FUNCTION_BLOCK Ps10Axis EXTENDS AxesBase
VAR_INPUT
END_VAR
VAR_OUTPUT
END_VAR
VAR
	{attribute 'OPC.UA.DA' := '0'}
	_config : Ps10OwisAxisConfig;
	{attribute 'OPC.UA.DA' := '0'}
	_coeAccess : CoeAccess;
	{attribute 'OPC.UA.DA' := '0'}
	_initConfigSerialCom : BOOL;	
	{attribute 'OPC.UA.DA' := '0'}
	_serialCom  : SerialCom(Prefix :='', Suffix := Const.CARRIAGE_RETURN);
	{attribute 'OPC.UA.DA' := '0'}
	_refSerialCom : REFERENCE TO SerialCom(Prefix :='', Suffix := Const.CARRIAGE_RETURN) := _serialCom;	 
	{attribute 'OPC.UA.DA' := '0'}
	_isReceived : BOOL;
	
	{attribute 'OPC.UA.DA' := '0'}
	_deliverMessages : INT;
	
	StatusMsg : STRING(255);
	AxisStatusMsg : STRING(255);
	DrivingCurrentMsg : STRING(255);
	HoldingCurrentMsg : STRING(255);
	LimitSwitchtMsg : STRING(255);
	ErrMsg : STRING(255);
	PositionMsg : STRING(255);
	CustomMsg : STRING(255);
	IsInMovingMsg : STRING(255);
	
	{region 'Commands'}	

	{attribute 'OPC.UA.DA' := '0'}
	_cmdConfigDeviceParameters : BOOL;
	{attribute 'OPC.UA.DA' := '0'}
	_cmdClearErr : BOOL;
	{attribute 'OPC.UA.DA' := '0'}
	_cmdMotorInit : BOOL;
	{attribute 'OPC.UA.DA' := '0'}
	_cmdDrivingCurrent : BOOL;
	{attribute 'OPC.UA.DA' := '0'}
	_cmdHoldingCurrent : BOOL;
	{attribute 'OPC.UA.DA' := '0'}	 
	_cmdLimitSwitch : BOOL;
	{attribute 'OPC.UA.DA' := '0'}
	_cmdReset : BOOL;
	{attribute 'OPC.UA.DA' := '0'}
	_cmdStopMotion : BOOL;		 
	{attribute 'OPC.UA.DA' := '0'}
	_cmdHomePosition : BOOL;
	{attribute 'OPC.UA.DA' := '0'}
	_cmdMoveAbsPosition : BOOL;
	{attribute 'OPC.UA.DA' := '0'}
	_customCmd : BOOL;
	{attribute 'OPC.UA.DA' := '0'}			  		   
	_cmdRaiseProperties : BOOL;	 
			
	{endregion}
		 
	{attribute 'OPC.UA.DA' := '0'}
	_initDevice : BOOL;	
		
	{attribute 'OPC.UA.DA' := '0'}
	_posToDegree : LREAL;
	{attribute 'OPC.UA.DA' := '0'}
	_cmd : STRING;
	{attribute 'OPC.UA.DA' := '0'}
	_itemScheduler : INT;
	{attribute 'OPC.UA.DA' := '0'}
	_itemRaisedProperties : INT;
	{attribute 'OPC.UA.DA' := '0'}
	_itemMove : INT;	
	{attribute 'OPC.UA.DA' := '0'}
	_itemInit : INT;
	{attribute 'OPC.UA.DA' := '0'}
	_itemdConfigDeviceParameters : INT;
	{attribute 'OPC.UA.DA' := '0'}
	_pulseGenerator : TON;
	{attribute 'OPC.UA.DA' := '0'}
	_pulseMoveGenerator : TON;	
	{attribute 'OPC.UA.DA' := '0'}
	_initPulseGenerator : TON;	
	{attribute 'OPC.UA.DA' := '0'}	
	_execPulseGenerator : TON;
	{attribute 'OPC.UA.DA' := '0'}	
	_configDeviceParamsPulseGenerator : TON;	
	
	{attribute 'OPC.UA.DA' := '0'}
	message : STRING;
	{attribute 'OPC.UA.DA' := '0'}
	lastMessage : STRING;	
	{attribute 'OPC.UA.DA' := '0'}
	stringLength : INT;
	{attribute 'OPC.UA.DA' := '0'}
	_convertDegreeToCount : LREAL := 83;
	{attribute 'OPC.UA.DA' := '0'}
	_currentAxisMode : STRING;
	{attribute 'OPC.UA.DA' := '0'}
	_currentPos : LREAL;	
	{attribute 'OPC.UA.DA' := '0'} 
	_currentPositionCounter : UINT;
	{attribute 'OPC.UA.DA' := '0'} 
	_isInMoving : BOOL;
END_VAR

IF NOT InitConfigSerialCom THEN
	ConfigureSerialCom();
ELSIF THIS^.Status = TExecutionState.Ready THEN				
	IF _refSerialCom.ErrorReceiveId = COMERROR_NOERROR THEN
		_refSerialCom(TxBuffer:= HardwareGlobalVariables.TxBufferFilterWheel, 
		 	      	  RxBuffer:= HardwareGlobalVariables.RxBufferFilterWheel);
	END_IF			

	// Init device	
	InitDevice();
		 				  	
	// Deliver messages
	IF _refSerialCom.IsReceived THEN		
		lastMessage := _refSerialCom.LastReceivedString;			
		stringLength := LEN(lastMessage);
		
		IF stringLength > 1 THEN
			message := LEFT(lastMessage, stringLength - 1);
		ELSE
			message := ' ';
		END_IF; 
				
		CASE _deliverMessages OF	
			EFeedbackMsgOwisPs10.AxisStateMsg :
				_currentAxisMode := MID(message, 1, STRING_TO_INT(AxesConst.AXIS_FILTER_WHEEL));
				AxisStatusMsg := ParseAxisStatus(_currentAxisMode);
			EFeedbackMsgOwisPs10.DrivingCurrentMsg :
				 DrivingCurrentMsg := message;
			EFeedbackMsgOwisPs10.HoldingCurrentMsg :
				 HoldingCurrentMsg := message;
			EFeedbackMsgOwisPs10.LimitSwitchMsg :
				 LimitSwitchtMsg := message;
			EFeedbackMsgOwisPs10.ErrMsg :
				 ErrMsg := message;
			EFeedbackMsgOwisPs10.PositionMsg :					
				_currentPos := STRING_TO_LREAL(message) / _convertDegreeToCount;
				PositionMsg := LREAL_TO_STRING(_currentPos);				
			EFeedbackMsgOwisPs10.CurrentPositionCounterMsg :
				_currentPositionCounter := STRING_TO_UINT(message);			
			EFeedbackMsgOwisPs10.CustomMsg :
				CustomMsg := message;						
			END_CASE
	END_IF		
			
	IF (_initDevice AND NOT _cmdClearErr AND NOT _cmdMotorInit AND NOT _cmdConfigDeviceParameters AND NOT _cmdDrivingCurrent AND NOT 
		_cmdHoldingCurrent AND NOT _cmdLimitSwitch AND NOT _cmdStopMotion AND NOT _cmdHomePosition AND NOT _cmdMoveAbsPosition AND NOT 
		_customCmd AND NOT _cmdRaiseProperties) THEN
			MessageScheduler();
	END_IF
	
	ConfigDeviceParameters(_cmdConfigDeviceParameters);
	ClearError(_cmdClearErr);
	MotorInit(_cmdMotorInit);
	SetDrivingCurrent(_cmdDrivingCurrent);
	SetHoldingCurrent(_cmdHoldingCurrent);
	SetLimitSwitch(_cmdLimitSwitch);
	Reset(_cmdReset);
	StopMotion(_cmdStopMotion);
	HomePosition(_cmdHomePosition);	
	MoveAbsPosition(_cmdMoveAbsPosition, _posToDegree);
	CustomCommand(_customCmd, _cmd);	
	RaisePropertiesChanged(_cmdRaiseProperties);	
	
END_IF

{attribute 'TcRpcEnable' := '1'}
METHOD ClearError
VAR_INPUT
	Execute : BOOL;
END_VAR
VAR
	cmd : STRING := 'ERRCLEAR';
END_VAR
IF Execute THEN
	_logger.Information(_message.Reset().Append(_config.Name).Append(' - Clear error').ToString());
	_serialCom.Send(cmd);	

	_cmdClearErr := FALSE;
END_IF
END_METHOD

METHOD ConfigDeviceParameters
VAR_INPUT
	Execute : BOOL;
END_VAR
VAR	
END_VAR
IF Execute THEN

	_cmdConfigDeviceParameters := TRUE;	

	IF _configDeviceParamsPulseGenerator.Q THEN
		_configDeviceParamsPulseGenerator(IN := FALSE, PT := T#10MS);
		
		CASE _itemdConfigDeviceParameters OF
			0:  _logger.Information(_message.Reset().Append(_config.Name).Append(' - Configure device parameters').ToString());
				_itemdConfigDeviceParameters := 1;				
								
			1: _cmdDrivingCurrent := TRUE;
				_itemdConfigDeviceParameters := 2;

			2: _cmdHoldingCurrent := TRUE;
				_itemdConfigDeviceParameters := 3;				
			
			3: _cmdLimitSwitch := TRUE;
				_itemdConfigDeviceParameters := 4;	
			
			4: _cmdMotorInit := TRUE;
				_itemdConfigDeviceParameters := 5;					
				
			5: _logger.Information(_message.Reset(). Append(_config.Name). Append(' - Configure device parameters done').ToString());	
			   _itemdConfigDeviceParameters := 0;			
			   _cmdConfigDeviceParameters := FALSE;
		END_CASE
	ELSE
		_configDeviceParamsPulseGenerator(IN := TRUE, PT := T#200MS);		
	END_IF		
END_IF
END_METHOD

METHOD ConfigureSerialCom
VAR_INPUT
END_VAR
IF _coeAccess.CoeOperation.Ready THEN
	_logger.Information(_message.Reset().Append('Start configuration com serial').ToString());
END_IF;	

_coeAccess.CoeOperation.Start();
_coeAccess(SerialCommunication := _config.SerialCommunication);
	
IF _coeAccess.CoeOperation.Done THEN
	_coeAccess.SetDone();	
 
	_Logger.Information(_message.Reset().
							Append('{').Append(TO_STRING(THIS^.Family)).Append('} : ').
							Append(' - Status : ').Append(TO_STRING(_coeAccess.Status)).ToString());	
	InitConfigSerialCom := TRUE;
END_IF
 
IF _coeAccess.CoeOperation.Error THEN	
	_coeAccess.SetError(0);
	
	_Logger.Error(_message.Reset().
							Append('{').Append(TO_STRING(THIS^.Family)).Append('} : ').
							Append(' - Status : ').Append(TO_STRING(_coeAccess.Status)).ToString());
	InitConfigSerialCom := TRUE;
END_IF

THIS^.Status := _coeAccess.Status;
State := _coeAccess.Status;
END_METHOD

{attribute 'TcRpcEnable' := '1'}
METHOD CustomCommand
VAR_INPUT
	Execute : BOOL;
	Cmd : STRING;
END_VAR
IF Execute THEN
	_logger.Information(_message.Reset().Append(_config.Name).Append(' - Custom : ').Append(Cmd).ToString());
	_deliverMessages := EFeedbackMsgOwisPs10.CustomMsg;									
	_serialCom.Send(Cmd);
	
	_customCmd := FALSE;
END_IF
END_METHOD

{attribute 'TcRpcEnable' := '1'}
METHOD ErrorMessages
VAR_INPUT
END_VAR
VAR
	cmd : STRING := '?MSG';
END_VAR
_deliverMessages := EFeedbackMsgOwisPs10.ErrMsg;	
_serialCom.Send(cmd);
END_METHOD

METHOD FB_init : BOOL
VAR_INPUT
	bInitRetains : BOOL; // if TRUE, the retain variables are initialized (warm start / cold start)
	bInCopyCode : BOOL;  // if TRUE, the instance afterwards gets moved into the copy code (online change)
	Config : Ps10OwisAxisConfig;
END_VAR
IF Config.IsEnabled THEN
	_config := Config;
	
	SUPER^._axisConfig.Name := Config.Name;
	SUPER^._axisConfig.DeviceID := Config.DeviceID;
	SUPER^._axisConfig.IsEnabled := Config.IsEnabled;
	SUPER^._axisConfig.LogLevel := Config.LogLevel;
	
	SUPER^.Name := Config.Name;
	SUPER^.DeviceID := Config.DeviceID;	
	THIS^.Family := DeviceFamily.Axes;
	
	_Logger.Information(_message.Reset().Append('Init ').
							Append('{').Append(TO_STRING(THIS^.Family)).Append('} - ').
							Append('{').Append(TO_STRING(Config.Name)).Append('}').ToString());																													
END_IF
END_METHOD

(** Axis state inquiry **)
METHOD GetAxisStatus : STRING
VAR_INPUT
END_VAR
VAR
	cmd : STRING := '?ASTAT';
END_VAR
_deliverMessages := EFeedbackMsgOwisPs10.AxisStateMsg;	
_serialCom.Send(cmd);
END_METHOD

(** Read out driving current with stepper motors in percent **)
METHOD PROTECTED GetDrivingCurrent
VAR_INPUT
END_VAR
VAR
	cmd : STRING := '?DRICUR';
END_VAR
_deliverMessages := EFeedbackMsgOwisPs10.DrivingCurrentMsg;	
_serialCom.Send(Concat(cmd, AxesConst.AXIS_FILTER_WHEEL));
END_METHOD

(** Read out holding current with stepper motor axis in percent **)
METHOD PROTECTED GetHoldingCurrent
VAR_INPUT
END_VAR
VAR
	cmd : STRING := '?HOLCUR';
END_VAR
_deliverMessages := EFeedbackMsgOwisPs10.HoldingCurrentMsg;	
_serialCom.Send(Concat(cmd, AxesConst.AXIS_FILTER_WHEEL));
END_METHOD

(** Read out limit switch mask for the axis **)
METHOD PROTECTED GetLimitSwitch
VAR_INPUT
END_VAR
VAR
	cmd : STRING := '?SMK';
END_VAR
_deliverMessages := EFeedbackMsgOwisPs10.LimitSwitchMsg;	
_serialCom.Send(Concat(cmd, AxesConst.AXIS_FILTER_WHEEL));
END_METHOD

(** Position Query **)
METHOD PROTECTED GetPosition
VAR_INPUT
END_VAR
VAR
	cmd : STRING := '?PSET';
END_VAR
_deliverMessages := EFeedbackMsgOwisPs10.PositionMsg;	
_serialCom.Send(Concat(cmd, AxesConst.AXIS_FILTER_WHEEL));
END_METHOD

{attribute 'TcRpcEnable' := '1'}
METHOD HomePosition
VAR_INPUT
	Execute : BOOL;
END_VAR
VAR
	cmd : STRING := 'REF';
END_VAR
IF Execute THEN	
	_logger.Information(_message.Reset().Append(_config.Name).Append(' - Home position : ').ToString());
	cmd := Concat(CONCAT(cmd, AxesConst.AXIS_FILTER_WHEEL), '=');	
	_serialCom.Send(Concat(cmd, '4'));
	
	_cmdHomePosition := FALSE;
END_IF
END_METHOD

PROPERTY InitConfigSerialCom : BOOL
GET
InitConfigSerialCom := _initConfigSerialCom;
END_GET
SET
_initConfigSerialCom := InitConfigSerialCom;
END_SET
END_PROPERTY

METHOD InitDevice
VAR_INPUT
END_VAR
VAR
	displayingPositionCmd : STRING := 'PWMSMODE';
	absoluteModeCmd : STRING := 'ABSOL';
	
	displayingPositionInDegree : STRING;
END_VAR
IF NOT _initDevice THEN	
	IF _initPulseGenerator.Q THEN
		_initPulseGenerator(IN := FALSE, PT := T#10MS);
		
		CASE _itemInit OF
			0:  _logger.Information(_message.Reset().Append(_config.Name).Append(' - InitDevice').ToString());
				_itemInit := 1;				
				
			1:  _cmdClearErr := TRUE;
				_itemInit := 2;
			
			2: // Absolute mode
				_serialCom.Send(CONCAT(absoluteModeCmd, AxesConst.AXIS_FILTER_WHEEL));	
				_itemInit := 10;
				
			10: _cmdConfigDeviceParameters := TRUE;	
			   _itemInit := 11;
			
			11: IF NOT _cmdConfigDeviceParameters THEN
					_itemInit := 20;
				END_IF
			
			20: GetAxisStatus();
				_itemInit := 21;
				
			21: // Displaying position in °
				displayingPositionInDegree := Concat(CONCAT(displayingPositionCmd, AxesConst.AXIS_FILTER_WHEEL), '=');
				_serialCom.Send(CONCAT(displayingPositionInDegree, '3'));				
				_itemInit := 22;													
				
			22:  IF _currentAxisMode = 'R' THEN	
					_itemInit := 30;	
				ELSE			
					_logger.Error(_message.Reset().Append(_config.Name).Append(' - Axis status : ').
								  Append(_currentAxisMode).ToString());
					_itemInit := 40;				  
			    END_IF							
				
			30:  GetPosition();
				_itemInit := 31;	
				
			31: _posToDegree := _currentPos;
				_itemInit := 40;
				
			40: _logger.Information(_message.Reset(). Append(_config.Name). Append(' - InitDevice done').ToString());	
				_itemInit := 0;			
				_initDevice	:= TRUE;
		END_CASE
	ELSE
		_initPulseGenerator(IN := TRUE, PT := T#100MS);		
	END_IF		
END_IF
END_METHOD

PROPERTY IsInMoving : bool
GET
IsInMoving := _isInMoving;
END_GET
SET
_isInMoving := IsInMoving;
END_SET
END_PROPERTY

METHOD MessageScheduler
VAR_INPUT
END_VAR
IF _pulseGenerator.Q THEN
	_pulseGenerator(IN := FALSE, PT := T#10MS);
	
	CASE _itemScheduler OF				
		0:	GetAxisStatus();
			_itemScheduler := 1;
						
		1:	GetPosition();
			_itemScheduler := 0;			
	END_CASE		
ELSE
	_pulseGenerator(IN := TRUE, PT := T#100MS);		
END_IF
END_METHOD

{attribute 'TcRpcEnable' := '1'}
METHOD MotorInit
VAR_INPUT
	Execute : BOOL;
END_VAR
VAR	
	cmd : STRING := 'INIT';
END_VAR
IF Execute THEN
	_logger.Information(_message.Reset().Append(_config.Name).Append(' - Enable the motor power stage').ToString());
	_serialCom.Send(Concat(cmd, AxesConst.AXIS_FILTER_WHEEL));	

	_cmdMotorInit := FALSE;	
END_IF
END_METHOD

{attribute 'TcRpcEnable' := '1'}
METHOD PROTECTED MoveAbsPosition 
VAR_INPUT
	Execute : BOOL;
	Position : LREAL;
END_VAR
VAR
	cmdSet : STRING := 'PSET';
	cmdGo : STRING := 'PGO';
	cmdCnt : STRING := '?CNT';
	cmd : STRING;	
END_VAR
IF Execute THEN

	_cmdMoveAbsPosition := TRUE;
	_posToDegree := Position;	
	
	IF _pulseMoveGenerator.Q THEN
		_pulseMoveGenerator(IN := FALSE, PT := T#10MS);
	
		CASE _itemMove OF
			0:	_logger.Information(_message.Reset().Append(_config.Name).Append(' - Move absolute position : ').
													 Append(TO_STRING(_posToDegree)).Append(' °').ToString());
								
				cmd := Concat(CONCAT(cmdSet, AxesConst.AXIS_FILTER_WHEEL), '=');				
				_serialCom.Send(CONCAT(cmd, LREAL_TO_STRING(_posToDegree * _convertDegreeToCount)));				
				_itemMove := 1;						
				
			1:  _serialCom.Send(Concat(cmdGo, AxesConst.AXIS_FILTER_WHEEL));											
				_itemMove := 2;	
				
			2:  _deliverMessages := EFeedbackMsgOwisPs10.CurrentPositionCounterMsg;	
				IF _currentPositionCounter <> (_posToDegree * _convertDegreeToCount) THEN					
					_serialCom.Send(Concat(cmdCnt, AxesConst.AXIS_FILTER_WHEEL));
					IsInMovingMsg := BOOL_TO_STRING(TRUE);	
				ELSE
					IsInMovingMsg := BOOL_TO_STRING(FALSE);	
					_itemMove := 3;	
				END_IF
								
			3: _cmdMoveAbsPosition := FALSE;
				_itemMove := 0;
			
		END_CASE			
	ELSE
		_pulseMoveGenerator(IN := TRUE, PT := T#100MS);	
	END_IF

END_IF
END_METHOD

METHOD PRIVATE ParseAxisStatus : STRING
VAR_INPUT
	CurrentAxisMode : STRING;
END_VAR
VAR
	Description : STRING;
END_VAR
IF CurrentAxisMode = 'I' THEN
	Description := 'Axis is not initialized';
ELSIF CurrentAxisMode = 'O' THEN
	Description := 'Axis is disabled';
ELSIF CurrentAxisMode = 'R' THEN
	Description := 'Axis initialized and ready';
ELSIF CurrentAxisMode = 'T' THEN
	Description := 'Axis is positioning in trapezoidal profile';
ELSIF CurrentAxisMode = 'V' THEN
	Description := 'Axis is operating in velocity mode';
ELSIF CurrentAxisMode = 'P' THEN
	Description := 'Reference motion is in progress';
ELSIF CurrentAxisMode = 'F' THEN
	Description := 'Axis is releasing a limit switch';
ELSIF CurrentAxisMode = 'L' THEN
	Description := 'Axis has been disabled after approaching a hardware limit switch(MINSTOP, MAXSTOP)';
ELSIF CurrentAxisMode = 'B' THEN
	Description := 'Aaxis has been stopped after approaching a brake switch(MINDEC, MAXDEC)';
ELSIF CurrentAxisMode = 'A' THEN
	Description := 'Axis has been disabled after limit switch error';
ELSIF CurrentAxisMode = 'M' THEN
	Description := 'Axis has been disabled after motion-controller error';
ELSIF CurrentAxisMode = 'Z' THEN
	Description := 'Axis has been disabled after timeout error';
ELSIF CurrentAxisMode = 'H' THEN
	Description := 'Phase initialization active (step motor axis)';
ELSIF CurrentAxisMode = 'U' THEN
	Description := 'Axis not enabled';
ELSIF CurrentAxisMode = 'E' THEN
	Description := 'Axis has been disabled after motion error';
ELSIF CurrentAxisMode = '?' THEN
	Description := 'Error, unknown state of axis';
ELSE
	Description := 'Unknown error';
END_IF

ParseAxisStatus := Description;
END_METHOD

{attribute 'TcRpcEnable' := '1'}
METHOD RaisePropertiesChanged
VAR_INPUT
	Execute : BOOL;
END_VAR
IF Execute THEN
	IF THIS^.Status <> TExecutionState.Ready THEN	
		_cmdRaiseProperties := FALSE;
		RETURN;
	END_IF	

	_cmdRaiseProperties := TRUE;
	
	IF _pulseGenerator.Q THEN
		_pulseGenerator(IN := FALSE, PT := T#10MS);	

		CASE _itemRaisedProperties OF
			0:  StateMsg := ' ';
				AxisStatusMsg := ' ';
				ErrMsg := ' ';
				PositionMsg := ' ';
				CustomMsg := ' ';
				
				_itemRaisedProperties := 10;
			
			10:  GetPosition();
				_itemRaisedProperties := 11;
			
			11:  GetAxisStatus();
				 _itemRaisedProperties := 12;
				 
			12:  ErrorMessages();
				 _itemRaisedProperties := 20;			
				 
			20:  _logger.Information(_message.Reset().Append(_config.Name).Append(' - PS10 Axis RaisePropertiesChanged').ToString());
				_cmdRaiseProperties := FALSE;				
				_itemRaisedProperties := 0;
			
		END_CASE
	ELSE
		_pulseGenerator(IN := TRUE, PT := T#100MS);	
	END_IF
END_IF
END_METHOD

{attribute 'TcRpcEnable' := '1'}
METHOD Reset
VAR_INPUT
	Execute : BOOL;
END_VAR
VAR
	cmd : STRING := 'RESETMB';
END_VAR
IF Execute THEN
	_logger.Information(_message.Reset().Append(_config.Name).Append(' - Release reset main board').ToString());
	_serialCom.Send(cmd);	
	
	_cmdReset := FALSE;
END_IF
END_METHOD

{attribute 'TcRpcEnable' := '1'}
METHOD SetDrivingCurrent
VAR_INPUT
	Execute : BOOL;
END_VAR
VAR
	cmdSet : STRING := 'DRICUR';
	cmd : STRING;
END_VAR
IF Execute THEN
	_logger.Information(_message.Reset().Append(_config.Name).Append(' - driving current with stepper motor: ').
		Append(TO_STRING(AxesConst.FW_DRIVING_CURRENT_IN_PERCENT)).ToString());
	
	cmd := Concat(CONCAT(cmdSet, AxesConst.AXIS_FILTER_WHEEL), '=');
	_serialCom.Send(CONCAT(cmd, TO_STRING(AxesConst.FW_DRIVING_CURRENT_IN_PERCENT)));	

	_cmdDrivingCurrent := FALSE;	
END_IF
END_METHOD

{attribute 'TcRpcEnable' := '1'}
METHOD SetHoldingCurrent
VAR_INPUT
	Execute : BOOL;
END_VAR
VAR
	cmdSet : STRING := 'HOLCUR';
	cmd : STRING;
END_VAR
IF Execute THEN
	_logger.Information(_message.Reset().Append(_config.Name).Append(' - holding current with stepper motor axes: ').
		Append(TO_STRING(AxesConst.FW_HOLDING_CURRENT_IN_PERCENT)).ToString());
	
	cmd := Concat(CONCAT(cmdSet, AxesConst.AXIS_FILTER_WHEEL), '=');
	_serialCom.Send(CONCAT(cmd, TO_STRING(AxesConst.FW_HOLDING_CURRENT_IN_PERCENT)));	

	_cmdHoldingCurrent := FALSE;	
END_IF
END_METHOD

{attribute 'TcRpcEnable' := '1'}
METHOD SetLimitSwitch
VAR_INPUT
	Execute : BOOL;
END_VAR
VAR
	cmdSet : STRING := 'SMK';
	cmd : STRING;
END_VAR
IF Execute THEN
	_logger.Information(_message.Reset().Append(_config.Name).Append(' -  limit switch mask for the axis: ').
		Append(TO_STRING(AxesConst.FW_LIMIT_SWITCH_MASK)).ToString());
	
	cmd := Concat(CONCAT(cmdSet, AxesConst.AXIS_FILTER_WHEEL), '=');
	_serialCom.Send(CONCAT(cmd, TO_STRING(AxesConst.FW_LIMIT_SWITCH_MASK)));	

	_cmdLimitSwitch := FALSE;	
END_IF
END_METHOD

{attribute 'TcRpcEnable' := '1'}
METHOD StopMotion
VAR_INPUT
	Execute : BOOL;
END_VAR
VAR
	cmd : STRING := 'STOP1';
END_VAR
IF Execute THEN	
	_logger.Information(_message.Reset().Append(_config.Name).Append(' - Stop motion').ToString());
	_serialCom.Send(cmd);
	
	_cmdStopMotion := FALSE;
END_IF
END_METHOD

END_FUNCTION_BLOCK

(* stored: Version 1.1.0.1, ProductVersion 3.1.4024.12
   POU Ps10Axis: Id {65318552-fa8a-4be4-9877-1eb5da08e2e6}, SpecialFunc None
   Folder Comamnds: Id {350d7b4c-9999-4614-8983-2b0788406443}
   Method ClearError: Id {9cf50f82-dedf-4020-a341-c2e03f9bd16b}
   Method ConfigDeviceParameters: Id {9dd7c1a3-38a3-4271-adf2-d5c1fd271f87}
   Method ConfigureSerialCom: Id {92ee4274-1822-4857-a351-1af2244cf04e}
   Method CustomCommand: Id {04426e00-f477-4383-857a-2ae2c5de4dbe}
   Method ErrorMessages: Id {af95c508-4de3-4b04-ad88-3fb38c9b4a6e}
   Method FB_init: Id {c9eecb17-8010-4deb-b770-2d445332fb7a}
   Method GetAxisStatus: Id {3fbf2da0-a10e-4662-ab0b-95ea943ad0ed}
   Method GetDrivingCurrent: Id {92b3f748-1524-4586-a2ca-ecd6e1233df8}
   Method GetHoldingCurrent: Id {1eac2e4b-31a7-47d1-83e9-91a91d90e56e}
   Method GetLimitSwitch: Id {d69a0b29-70d3-44d2-b788-e7ab365eced6}
   Method GetPosition: Id {55a3b673-e715-4d70-9fa7-5225e4770e89}
   Method HomePosition: Id {142d51a5-57ef-4f7b-b18a-4cfaf2920b91}
   Property InitConfigSerialCom: Id {2aa5b88d-df39-4f9b-949f-1e8e44a662c9}
   Get Get: Id {494cec2c-0a6e-4e21-8cea-50ca2358b100}
   Set Set: Id {5729c6bb-be11-4151-8251-605ad3510059}
   Method InitDevice: Id {5c2fcf27-05f4-4bb9-9c40-55e9bc5563c8}
   Property IsInMoving: Id {43f5a690-3f81-4021-9bd2-2250a324fef6}
   Get Get: Id {43b5b94b-ba0a-4053-90d8-b0b48186412a}
   Set Set: Id {5eefe730-1f7f-423f-84ac-5e9df6527cc9}
   Method MessageScheduler: Id {d15cb2a3-cb63-4708-a63c-d14e3c192308}
   Method MotorInit: Id {9d90297e-68a2-4beb-b5a0-edfb71b5534e}
   Method MoveAbsPosition: Id {e52af445-02be-4345-a161-7a76bf74adb8}
   Method ParseAxisStatus: Id {2ff9b0bb-a1ce-404f-9822-774a93978c34}
   Method RaisePropertiesChanged: Id {45cfc383-769d-41a8-b977-b8e03a3eabf9}
   Method Reset: Id {01c8b468-ecb2-466c-944f-2e53330ceefa}
   Method SetDrivingCurrent: Id {27024876-06ae-4839-8285-7cc84996afd3}
   Method SetHoldingCurrent: Id {d857ec78-2ed8-4b2a-9270-7cf05b795f2c}
   Method SetLimitSwitch: Id {f83492f6-17f2-404b-ad6a-1bc3f26ce477}
   Method StopMotion: Id {f85cc7d7-3ac6-41e1-8df5-12989e0bdb2e} *)
